PROGRAM PLC_PRG
VAR
	//Visualisation buttons	
	mxButtonReset	: BOOL;	
	mxButtonStart: BOOL;

	//Internal use
	mxStart: BOOL;
	mxDone: BOOL;
	mxComBusy: BOOL;
	CommData: CommunicationData;	
	
	//Motion Function Blocks
	fbCommunicator: Communicator;
	fbABBGoToHome_1: ABBGoToHome;
	fbABBGoToTable_1: ABBGoToTable;
END_VAR

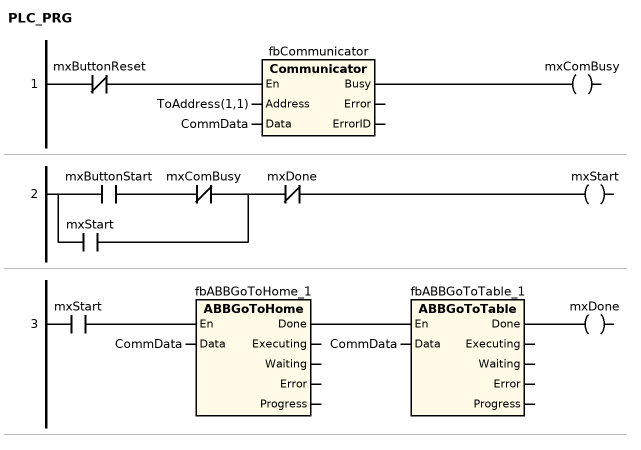
// NETWORK 1
fbCommunicator(En := NOT mxButtonReset, Address := ToAddress(1,1), Data := CommData); // Communicator
mxComBusy := fbCommunicator.Busy;

// NETWORK 2
mxStart := (mxButtonStart AND NOT mxComBusy OR mxStart) AND NOT mxDone;

// NETWORK 3
fbABBGoToHome_1(En := mxStart, Data := CommData); // ABBGoToHome
fbABBGoToTable_1(En := fbABBGoToHome_1.Done, Data := CommData); // ABBGoToTable
mxDone := fbABBGoToTable_1.Done;

END_PROGRAM

(* stored: Version 1.1.0.1, ProductVersion 3.1.4022.12
   POU PLC_PRG: Id {3ddf41dd-5784-480c-987d-9d96251b8aa6}, SpecialFunc None *)
